FUNCTION_BLOCK SPLIT_AB_INTO_AX (* this Function splits the 8 AX (BOOL) adapters from a AB (BYTE) *)
  (* Standard: 61499-2; Description: Copyright (c) 2026 Meisterschulen am Ostbahnhof SPDX-License-Identifier: EPL-2.0 *)
  (* Version 1.0, 2026-03-05, Franz Höpfinger, Meisterschulen am Ostbahnhof, initial API and implementation and/or initial documentation *)
  PACKAGE adapter::splitting;
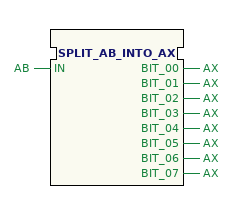
  SOCKETS
    IN : adapter::types::unidirectional::AB; (* BYTE Input *)
  END_SOCKETS
  PLUGS
    BIT_00 : adapter::types::unidirectional::AX; (* Bool Bit 0 *)
    BIT_01 : adapter::types::unidirectional::AX; (* Bool Bit 1 *)
    BIT_02 : adapter::types::unidirectional::AX; (* Bool Bit 2 *)
    BIT_03 : adapter::types::unidirectional::AX; (* Bool Bit 3 *)
    BIT_04 : adapter::types::unidirectional::AX; (* Bool Bit 4 *)
    BIT_05 : adapter::types::unidirectional::AX; (* Bool Bit 5 *)
    BIT_06 : adapter::types::unidirectional::AX; (* Bool Bit 6 *)
    BIT_07 : adapter::types::unidirectional::AX; (* Bool Bit 7 *)
  END_PLUGS
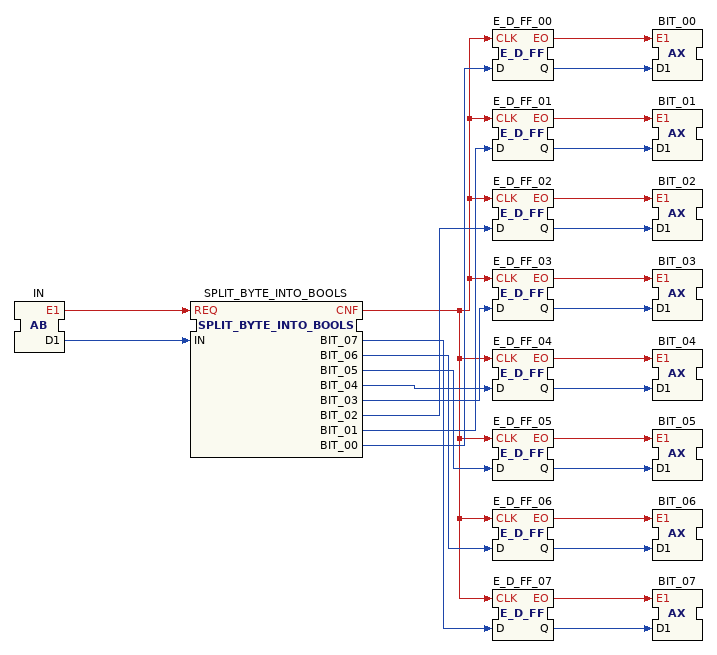
  FBS
    E_D_FF_00 : iec61499::events::E_D_FF;
    E_D_FF_01 : iec61499::events::E_D_FF;
    E_D_FF_02 : iec61499::events::E_D_FF;
    E_D_FF_03 : iec61499::events::E_D_FF;
    E_D_FF_04 : iec61499::events::E_D_FF;
    E_D_FF_05 : iec61499::events::E_D_FF;
    E_D_FF_06 : iec61499::events::E_D_FF;
    E_D_FF_07 : iec61499::events::E_D_FF;
    SPLIT_BYTE_INTO_BOOLS : eclipse4diac::utils::splitting::SPLIT_BYTE_INTO_BOOLS;
  END_FBS
  EVENT_CONNECTIONS
    IN.E1 TO SPLIT_BYTE_INTO_BOOLS.REQ;
    SPLIT_BYTE_INTO_BOOLS.CNF TO E_D_FF_00.CLK;
    SPLIT_BYTE_INTO_BOOLS.CNF TO E_D_FF_01.CLK;
    SPLIT_BYTE_INTO_BOOLS.CNF TO E_D_FF_02.CLK;
    SPLIT_BYTE_INTO_BOOLS.CNF TO E_D_FF_03.CLK;
    SPLIT_BYTE_INTO_BOOLS.CNF TO E_D_FF_04.CLK;
    SPLIT_BYTE_INTO_BOOLS.CNF TO E_D_FF_05.CLK;
    SPLIT_BYTE_INTO_BOOLS.CNF TO E_D_FF_06.CLK;
    SPLIT_BYTE_INTO_BOOLS.CNF TO E_D_FF_07.CLK;
    E_D_FF_00.EO TO BIT_00.E1;
    E_D_FF_01.EO TO BIT_01.E1;
    E_D_FF_02.EO TO BIT_02.E1;
    E_D_FF_03.EO TO BIT_03.E1;
    E_D_FF_04.EO TO BIT_04.E1;
    E_D_FF_05.EO TO BIT_05.E1;
    E_D_FF_06.EO TO BIT_06.E1;
    E_D_FF_07.EO TO BIT_07.E1;
  END_CONNECTIONS
  DATA_CONNECTIONS
    IN.D1 TO SPLIT_BYTE_INTO_BOOLS.IN;
    SPLIT_BYTE_INTO_BOOLS.BIT_07 TO E_D_FF_07.D;
    SPLIT_BYTE_INTO_BOOLS.BIT_06 TO E_D_FF_06.D;
    SPLIT_BYTE_INTO_BOOLS.BIT_05 TO E_D_FF_05.D;
    SPLIT_BYTE_INTO_BOOLS.BIT_04 TO E_D_FF_04.D;
    SPLIT_BYTE_INTO_BOOLS.BIT_03 TO E_D_FF_03.D;
    SPLIT_BYTE_INTO_BOOLS.BIT_02 TO E_D_FF_02.D;
    SPLIT_BYTE_INTO_BOOLS.BIT_01 TO E_D_FF_01.D;
    SPLIT_BYTE_INTO_BOOLS.BIT_00 TO E_D_FF_00.D;
    E_D_FF_00.Q TO BIT_00.D1;
    E_D_FF_01.Q TO BIT_01.D1;
    E_D_FF_02.Q TO BIT_02.D1;
    E_D_FF_03.Q TO BIT_03.D1;
    E_D_FF_04.Q TO BIT_04.D1;
    E_D_FF_05.Q TO BIT_05.D1;
    E_D_FF_06.Q TO BIT_06.D1;
    E_D_FF_07.Q TO BIT_07.D1;
  END_CONNECTIONS
END_FUNCTION_BLOCK
